(* CoDeSys 2.3 export: BATCHERCLASS.EXP *)

(* Data type in ENUM *)
TYPE BatcherClass : (Capacity:=1, Flow, Weight);
END_TYPE
